FUNCTION_BLOCK FB_AlarmManager
VAR_INPUT
END_VAR
VAR_OUTPUT
	aAlarmBuffer			: ARRAY[1..25] OF ST_Alarm;
END_VAR
VAR PERSISTENT
	aAlarmHistory			: ARRAY[1..100] OF ST_Alarm;
END_VAR
VAR
	nAlarmBufferSize		: USINT := 25;
	nAlarmHistorySize 		: USINT := 100;
END_VAR

METHOD M_Add : BOOL
VAR_INPUT
	nAlarmPriority		: USINT;
	sErrorMsg 			: STRING(50);
END_VAR
VAR
	nItem				: USINT;
	nIndex				: USINT := 1;
	stNewAlarm			: ST_Alarm;
	stTempAlarm_1		: ST_Alarm;
	stTempAlarm_2		: ST_Alarm;
END_VAR
// store new alarm into ST_Alarm format
stNewAlarm.nAlarmPriority := nAlarmPriority;
stNewAlarm.sErrorMsg := sErrorMsg;
// stNewAlarm.dtDateAndTime := Tc2_Utilities.SYSTEMTIME_TO_DT;

// store new alarm at top of buffer
stTempAlarm_1 := aAlarmBuffer[1];
aAlarmBuffer[1] := stNewAlarm;
nIndex := 2;

// move all older alarms down
WHILE ((aAlarmBuffer[nItem].sErrorMsg <> '') AND (nIndex < 25)) DO
	stTempAlarm_2 := aAlarmBuffer[nIndex];
	aAlarmBuffer[nIndex] := stTempAlarm_1;
	stTempAlarm_1 := stTempAlarm_2;
	nIndex := nIndex + 1;
END_WHILE
END_METHOD

METHOD M_Dismiss : BOOL
VAR_INPUT
END_VAR
END_METHOD

END_FUNCTION_BLOCK

(* stored: Version 1.1.0.1, ProductVersion 3.1.4024.11
   POU FB_AlarmManager: Id {c5be2f96-c55a-41d0-80c3-baa0954f0294}, SpecialFunc None
   Method M_Add: Id {16147c9d-b68e-4b50-8ed2-44a0cdd145f8}
   Method M_Dismiss: Id {eb7ebf00-dc70-4154-b77c-67f0ce25e28a} *)
